FUNCTION_BLOCK FB_MqttLightDiscovery EXTENDS FB_MqttDeviceDiscoveryBase
VAR_INPUT
END_VAR
VAR_OUTPUT
END_VAR
VAR
	stConfig : ST_MqttLightConfiguration;
END_VAR

PROPERTY PROTECTED Component : STRING(30)
GET
Component := 'light';
END_GET
END_PROPERTY

METHOD  ConfigToJson : STRING(1000)
VAR_INPUT
END_VAR
VAR
	fbJsonWriter : FB_JsonSaxWriter;
END_VAR
fbJsonWriter.ResetDocument();
fbJsonWriter.StartObject();
fbJsonWriter.AddKeyString(key := 'cmd_t', value := stConfig.command_topic);
fbJsonWriter.AddKeyString(key := 'stat_t', value := stConfig.state_topic);
fbJsonWriter.AddKeyString(key := 'uniq_id', value := stConfig.unique_id);
fbJsonWriter.AddKeyString(key := 'name', value := stConfig.name);
THIS^.DevInfoToJson(rJsonWriter := fbJsonWriter);
fbJsonWriter.EndObject();
fbJsonWriter.CopyDocument(pDoc := ConfigToJson, nDoc := 1000);
END_METHOD

PROPERTY Configuration : ST_MqttLightConfiguration
GET
Configuration := THIS^.stConfig;
END_GET
SET
this^.stConfig := Configuration;
END_SET
END_PROPERTY

END_FUNCTION_BLOCK

(* stored: Version 1.1.0.1, ProductVersion 3.1.4024.5
   POU FB_MqttLightDiscovery: Id {e838779f-4c08-477f-aa69-fe0c4f3677af}, SpecialFunc None
   Property Component: Id {890d4baf-9b7c-45f1-9eb6-e6dd064d139f}
   Get Get: Id {b8d496a3-2e5a-418a-99c8-0afea46ea387}
   Method ConfigToJson: Id {dd60e862-3412-40fb-8713-20da07d4089e}
   Property Configuration: Id {28606575-3785-46d2-b1d7-ca887d660ce1}
   Get Get: Id {3e3bc15d-64d9-4969-8d21-38ab9b86f779}
   Set Set: Id {81793631-04d3-4bdf-8628-0078c8095124} *)
